FUNCTION_BLOCK FB_Dispenser
VAR_INPUT
	bSens1 : BOOL;
	bSens2 : BOOL;
	bSens3 : BOOL;
	
	bEnable : BOOL;
	bExecute : BOOL;
	
END_VAR
VAR_OUTPUT
	Schnecke1 : BOOL;
	Schnecke2 : BOOL;
	Schnecke3 : BOOL;
END_VAR
VAR
END_VAR

Schnecke1 := FALSE;
Schnecke2 := FALSE;
Schnecke3 := FALSE;

IF bSens1 AND bEnable AND bExecute THEN
	Schnecke1 := TRUE;
	
ELSIF bSens2 AND bEnable AND bExecute THEN
	Schnecke2 := TRUE;
	
ELSIF bSens3 AND bEnable AND bExecute THEN
	Schnecke3 := TRUE;
	
END_IF

END_FUNCTION_BLOCK

(* stored: Version 1.1.0.1
   POU FB_Dispenser: Id {69835d49-650a-4d96-b161-fd36406bf87d}, SpecialFunc None *)
